# EPICS IOC start-up script: iocBoot/iocoh26/settings.iocsh
# IOC Name
epicsEnvSet("IOC", "iocoh26")

# Shell prompt
epicsEnvSet("IOCSH_PS1", "$(IOC)> ")

# prefix used for all PVs in this IOC
epicsEnvSet("PREFIX", "oh26:")

#For devIocStats
epicsEnvSet("ENGINEER", "nmarks")
epicsEnvSet("LOCATION", "$(HOSTNAME=location)")
epicsEnvSet("GROUP", "BC")

# search path for database files
epicsEnvSet("EPICS_DB_INCLUDE_PATH", ".")

# search path for streamDevice protocol files
epicsEnvSet("STREAM_PROTOCOL_PATH", ".")

# search path for lua scripts
epicsEnvSet("LUA_SCRIPT_PATH", "./lua")

# Specify largest array CA will transport
# Note for N doubles, need N*8 bytes+some overhead
epicsEnvSet("EPICS_CA_MAX_ARRAY_BYTES", 64010)
